(* IEC 61131-3 sources: conversion/test/times, 4 files *)

(* ---- LDateAndTimeToSimotionDateToD.st ---- *)
NAMESPACE Simatic.Ax.Conversion.Times

    {TestFixture}
    CLASS TestLDateAndTimeToSimotionDateTime

        {Test}
        METHOD PUBLIC CheckStartTime
            //test with 1ms added from initial time
            VAR_TEMP
                inputTimestamp : LDATE_AND_TIME := LDT#1992-01-01-00:00:00.001;
                simotionDate : DWORD;
                simotionTime : DWORD;
            END_VAR
            LDateAndTimeToSimotionDateTime(inputTimestamp, simotionTime, simotionDate);
            AxUnit.Assert.Equal(simotionTime , DWORD#1);
            AxUnit.Assert.Equal(simotionDate , DWORD#1);
        END_METHOD

        {Test}
        METHOD PUBLIC CheckCurrentTime
            VAR_TEMP
                inputTimestamp : LDATE_AND_TIME := LDT#2023-10-31-15:57:03.483;
                simotionDate : DWORD;
                simotionTime : DWORD;
            END_VAR

            LDateAndTimeToSimotionDateTime(SimaticTime := inputTimestamp, simotionTime => simotionTime, simotionDate => simotionDate);
            //the values have been read from a simotion plc and converted, so they proven to be valid
            AxUnit.Assert.Equal(simotionTime , DWORD#57423483);
            AxUnit.Assert.Equal(simotionDate , DWORD#11627);

        END_METHOD

    END_CLASS

END_NAMESPACE

(* ---- SimotionDateToDToLDateAndTime.st ---- *)
NAMESPACE Simatic.Ax.Conversion.Times

    {TestFixture}
    CLASS TestSimotionDateTimeToLDateAndTime

        {Test}
        METHOD PUBLIC CheckStartTime
            //test with 1ms added from initial time
            VAR_TEMP
                timestamp : LDATE_AND_TIME;
                simotionDate : DWORD := DWORD#1;
                simotionTime : DWORD := DWORD#1;
            END_VAR
            timestamp := SimotionDateTimeToLDateAndTime(SimotionTime := simotionTime, SimotionDate := simotionDate);
            AxUnit.Assert.Equal(timestamp = LDATE_AND_TIME#1992-01-01-00:00:00.001, TRUE);
        END_METHOD

        {Test}
        METHOD PUBLIC CheckCurrentTime
            VAR_TEMP
                timestamp : LDATE_AND_TIME;
                simotionDate : DWORD := DWORD#11627;
                simotionTime : DWORD := DWORD#57423483;
            END_VAR
            timestamp := SimotionDateTimeToLDateAndTime(SimotionTime := simotionTime, SimotionDate := simotionDate);
            //the values have been read from a simotion plc and converted, so they proven to be valid
            AxUnit.Assert.Equal(timestamp = LDT#2023-10-31-15:57:03.483, TRUE);

        END_METHOD

    END_CLASS

END_NAMESPACE

(* ---- ToLDateAndTime.st ---- *)
NAMESPACE Simatic.Ax.Conversion.Times

    {TestFixture}
    CLASS TestSimotionDateTimeToLDateAndTime

        {Test}
        METHOD PUBLIC CheckStartTime
            //test with 1ms added from initial time
            VAR_TEMP
                timestamp : LDATE_AND_TIME;
                SimotionDateTime : SimotionDateTime;
            END_VAR
            SimotionDateTime.SimotionDate := DWORD#1;
            SimotionDateTime.SimotionTime := DWORD#1;
            timestamp := SToLDateAndTime(SimotionDateTime);
            AxUnit.Assert.Equal(timestamp = LDATE_AND_TIME#1992-01-01-00:00:00.001, TRUE);
        END_METHOD

        {Test}
        METHOD PUBLIC CheckCurrentTime
            VAR_TEMP
                timestamp : LDATE_AND_TIME;
                SimotionDateTime : SimotionDateTime;
            END_VAR
            SimotionDateTime.SimotionDate := DWORD#11627;
            SimotionDateTime.SimotionTime := DWORD#57423483;
            timestamp := SToLDateAndTime(SimotionDateTime);
            //the values have been read from a simotion plc and converted, so they proven to be valid
            AxUnit.Assert.Equal(timestamp = LDT#2023-10-31-15:57:03.483, TRUE);

        END_METHOD

    END_CLASS

END_NAMESPACE

(* ---- ToSimotionDateTime.st ---- *)
NAMESPACE Simatic.Ax.Conversion.Times

    {TestFixture}
    CLASS TestLDateAndTimeToSimotionDateTime

        {Test}
        METHOD PUBLIC CheckStartTime
            //test with 1ms added from initial time
            VAR_TEMP
                inputTimestamp : LDATE_AND_TIME := LDT#1992-01-01-00:00:00.001;
                retval : SimotionDateTime;
                simotionDate : DWORD;
                simotionTime : DWORD;
            END_VAR
            retval := ToSimotionDateTime(inputTimestamp);
            AxUnit.Assert.Equal(retval.simotionTime , DWORD#1);
            AxUnit.Assert.Equal(retval.simotionDate , DWORD#1);
        END_METHOD

        {Test}
        METHOD PUBLIC CheckCurrentTime
            VAR_TEMP
                inputTimestamp : LDATE_AND_TIME := LDT#2023-10-31-15:57:03.483;
                retval : SimotionDateTime;
            END_VAR

            retval := ToSimotionDateTime(inputTimestamp);
            //the values have been read from a simotion plc and converted, so they proven to be valid
            AxUnit.Assert.Equal(retval.SimotionTime , DWORD#57423483);
            AxUnit.Assert.Equal(retval.SimotionDate , DWORD#11627);

        END_METHOD

    END_CLASS

END_NAMESPACE
